// TIA Portal V17 export
// export: Created 2024-09-02T12:50:04.9130735Z, ExportSetting WithDefaults, DisplayName Totally Integrated Automation Portal, DisplayVersion V17, DisplayName TIA Portal Openness, DisplayVersion V17, DisplayName TIA Portal Version Control Interface, DisplayVersion V17, DisplayName STEP 7 Professional, DisplayVersion V17, DisplayName STEP 7 Safety, DisplayVersion V17, DisplayName WinCC Professional, DisplayVersion V17
DATA_BLOCK "GraDB_Home"   // DB175
{ S7_Optimized_Access := 'TRUE'; DB_Accessible_From_OPC_UA := 'FALSE' }
AUTHOR : VAF
FAMILY : SK
NAME : SK
VERSION : 0.1
// stored: AutoNumber false, DBAccessibleFromOPCUA false, IsOnlyStoredInLoadMemory false, IsRetainMemResEnabled false, IsWriteProtectedInAS false, MemoryReserve 0
   VAR
      noAction : Bool;
      OP70_1 : Struct
         Home_SK : Bool;   // Grundstellung Schrittkette / Basic position Step chain
         Finished : Bool := false;   // Fertigmeldung / Finished message
      END_STRUCT;
      OP70_2 : Struct
         Home_SK : Bool;   // Grundstellung Schrittkette / Basic position Step chain
         Finished : Bool := false;   // Fertigmeldung / Finished message
      END_STRUCT;
   END_VAR
BEGIN
END_DATA_BLOCK
